(* Schneider Machine Expert - Basic project PLC, file version 2.7.0.0 *)
(* ProjectInformations: Name=New project *)

HARDWARE
  Cpu 0: TM221CE16R
  EthernetConfiguration: NetworkName=M221, IpAllocationMode=FixedAddress, IpAddress=0.0.0.0, SubnetMask=0.0.0.0
  SerialLineConfiguration: Baud=Baud9600, Parity=ParityNone, DataBits=DataBits8, StopBits=StopBits1, PhysicalMedium=PhysicalMediumRs485, TransmissionMode=TransmissionModeModbusRtu, SlaveId=1, Addressing=SlaveAddressing
  MastTask: UsePeriodScanMode=false, PeriodScan=100
  FastTask: Period=255
  CpuBehavior: StartingMode=StartAsPreviousState, AutoSaveRamOnEeprom=true, WatchdogPeriod=250

SYMBOLS  (address, symbol, comment, settings)
  %M1         "Detect Kereta"
  %M2         "Start Lub"
  %M3         "Stop Lub"
  %M4         "Servo Reverse"
  %M5         "Starter Loop"
  %M6         "Stopper Loop"
  %TM0        "Proximity Delay"  [Preset=30, Base=OneSecond]
  %TM1        "Lub Timer"  [Preset=5000, Base=OneMilliSeconds, IsDynamicPreset=true]
  %TM2        "Retract Delay"  [Preset=3, Base=OneSecond]
  %TM3        "Timer Reverse"  [Preset=6, Base=OneMilliSeconds]
  %I0.0       "Proximity"
  %I0.1       "Oil Level Low"
  %I0.2       "Pressure High"
  %Q0.0       "Lubricator"
  %Q0.1       "Buzzer Oil Level"
  %Q0.2       "Buzzer Pressure"
  %Q0.4       "Forward"
  %Q0.5       "Reverse"

POU New POU
  (* SectionNumber=1 *)

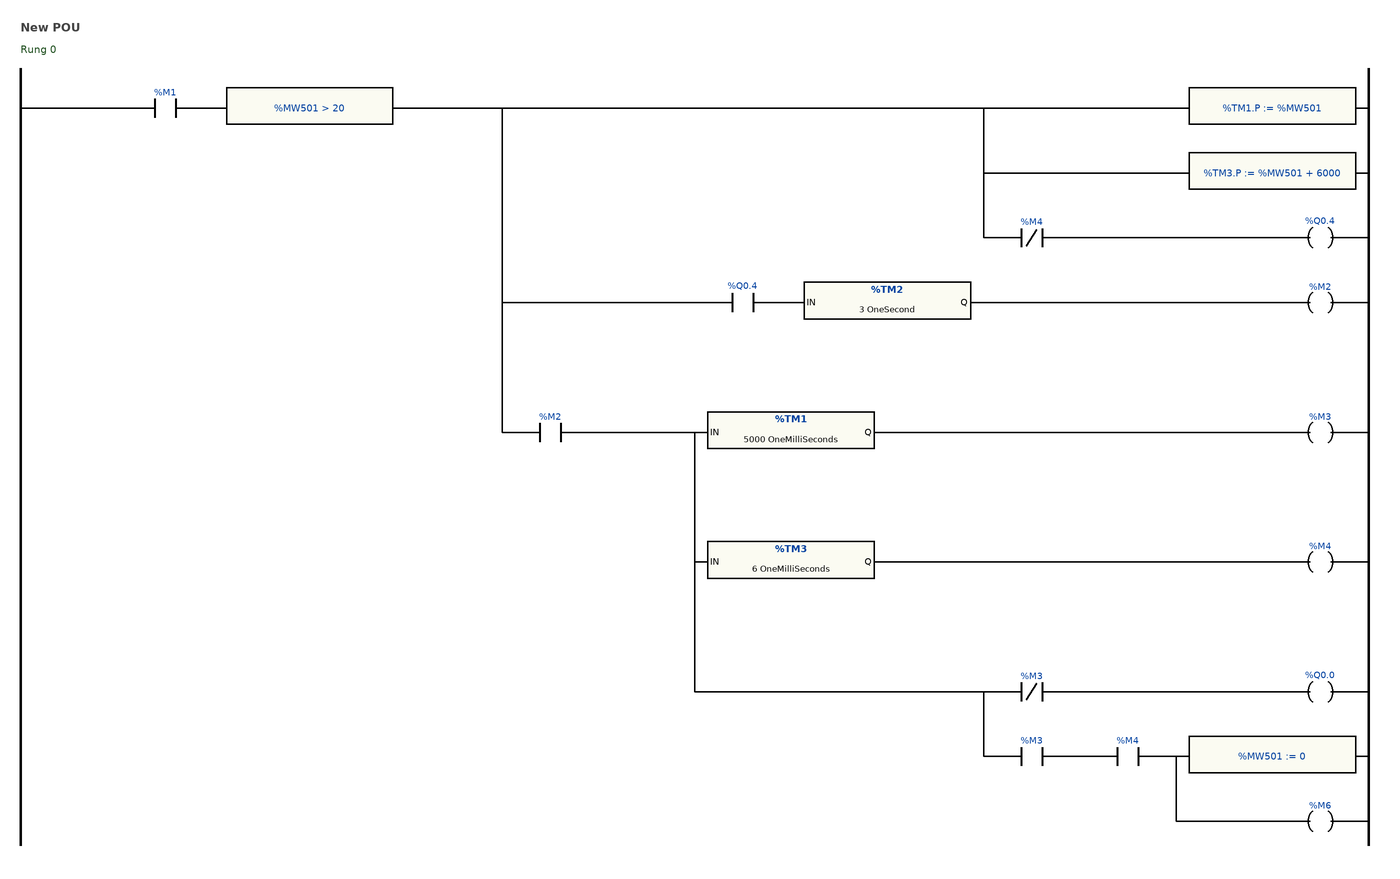

// Rung 0
  LD 1
  MULTIFB
  LD 1
  AND %M1
  AND [ %MW501 > 20 ]
  ST %MW2009:X0
  LD %MW2009:X0
  MPS
  [ %TM1.P := %MW501 ]
  MRD
  [ %TM3.P := %MW501 + 6000 ]
  MPP
  ANDN %M4
  ST %Q0.4
  BLK %TM2
  LD %MW2009:X0
  AND %Q0.4
  IN
  OUT_BLK
  LD Q
  ST %M2
  END_BLK
  LD %MW2009:X0
  AND %M2
  ST %MW2009:X1
  BLK %TM1
  LD %MW2009:X1
  IN
  OUT_BLK
  LD Q
  ST %M3
  END_BLK
  BLK %TM3
  LD %MW2009:X1
  IN
  OUT_BLK
  LD Q
  ST %M4
  END_BLK
  LD %MW2009:X1
  MPS
  ANDN %M3
  ST %Q0.0
  MPP
  AND %M3
  AND %M4
  [ %MW501 := 0 ]
  ST %M6
  MULTIFB
  // as ST:
  //   IF %M1 AND %MW501 > 20 THEN %TM1.P := %MW501; END_IF;
  //   IF %M1 AND %MW501 > 20 THEN %TM3.P := %MW501 + 6000; END_IF;
  //   %Q0.4 := %M1 AND %MW501 > 20 AND NOT %M4;
  //   %TM2(IN := %M1 AND %MW501 > 20 AND %Q0.4);
  //   %M2 := %TM2.Q;
  //   %TM1(IN := %M1 AND %MW501 > 20 AND %M2);
  //   %M3 := %TM1.Q;
  //   %TM3(IN := %M1 AND %MW501 > 20 AND %M2);
  //   %M4 := %TM3.Q;
  //   %Q0.0 := %M1 AND %MW501 > 20 AND %M2 AND NOT %M3;
  //   _t1 := %M1 AND %MW501 > 20 AND %M2 AND %M3 AND %M4;
  //   IF _t1 THEN %MW501 := 0; END_IF;
  //   %M6 := _t1;

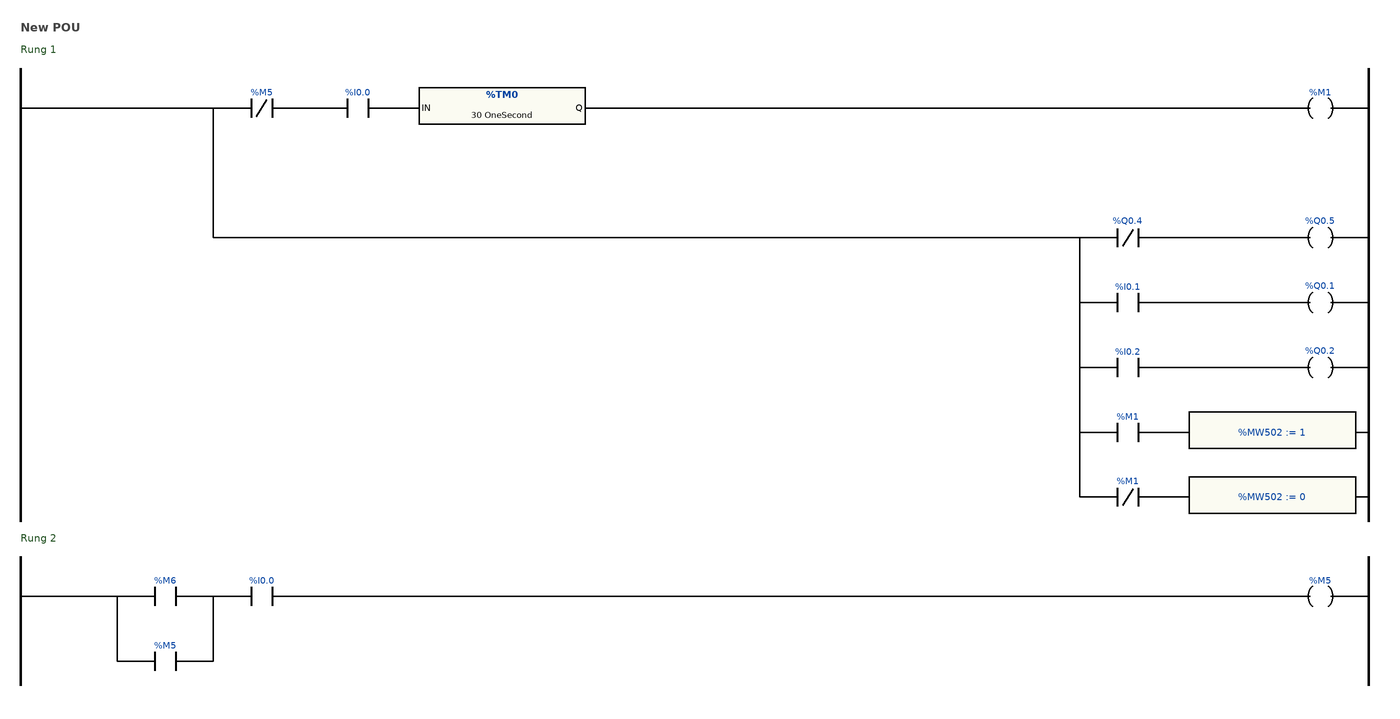

// Rung 1
  LD 1
  MULTIFB
  LD 1
  ST %MW2009:X0
  BLK %TM0
  LD %MW2009:X0
  ANDN %M5
  AND %I0.0
  IN
  OUT_BLK
  LD Q
  ST %M1
  END_BLK
  LD %MW2009:X0
  MPS
  ANDN %Q0.4
  ST %Q0.5
  MRD
  AND %I0.1
  ST %Q0.1
  MRD
  AND %I0.2
  ST %Q0.2
  MRD
  AND %M1
  [ %MW502 := 1 ]
  MPP
  ANDN %M1
  [ %MW502 := 0 ]
  MULTIFB
  // as ST:
  //   %TM0(IN := NOT %M5 AND %I0.0);
  //   %M1 := %TM0.Q;
  //   %Q0.5 := NOT %Q0.4;
  //   %Q0.1 := %I0.1;
  //   %Q0.2 := %I0.2;
  //   IF %M1 THEN %MW502 := 1; END_IF;
  //   IF NOT %M1 THEN %MW502 := 0; END_IF;

// Rung 2
  LD 1
  AND( %M6
  OR %M5
  )
  AND %I0.0
  ST %M5
  // as ST:
  //   %M5 := (%M6 OR %M5) AND %I0.0;
